PROGRAM MAIN
VAR
	VarOut AT %Q*: BOOL;
	VarIn AT %I*: BOOL;
END_VAR

VarOut := VarIn;

END_PROGRAM

(* stored: Version 1.1.0.1, ProductVersion 3.1.4024.5
   POU MAIN: Id {265004ad-ee78-4b56-a154-346e846c21bb}, SpecialFunc None *)
